TYPE ST_MESSAGE_CTRL :
STRUCT
  Cmd         : E_MESSAGE_CTRL;
END_STRUCT
END_TYPE

(* stored: Version 1.1.0.1, ProductVersion 3.1.4026.20
   DUT ST_MESSAGE_CTRL: Id {4b2b61d2-038a-439f-9446-6e8671ba15fd} *)
